Staubli VAL3: AXIS8.pjx

--- AXIS8.pjx ---
Parameters version=s7.2.1 stackSize=5000 millimeterUnit=true
Program file=del.pgx
Program file=find.pgx
Program file=findValue.pgx
Program file=get.pgx
Program file=getSize.pgx
Program file=getType.pgx
Program file=getValue.pgx
Program file=getVelocity.pgx
Program file=loadCycle.pgx
Program file=new.pgx
Program file=onEdit.pgx
Program file=onInsert.pgx
Program file=onProgEnd.pgx
Program file=onRun.pgx
Program file=onStart.pgx
Program file=onStop.pgx
Program file=set.pgx
Program file=setValue.pgx
Program file=setVelocity.pgx
Data file=AXIS8.dtx
Library alias=language path=Disk://kernel/language/language.pjx
Library alias=use path=Disk://kernel/userPage/userPage.pjx

--- AXIS8.dtx ---
num i = 6
public num nSaveaxis = 17746
public num nSaveaxis1 = 55156
public num nVelocity = 8
string l_sItem = "workPos"
public string sItems
public string sSaveaxis = "workPos"
public bool bAxisRun
public aio MbAI_a8Axispose = {link=ModbusSrv-0\Modbus-Word\MbAI_a8Axispose}
public aio MbAI_aCurPosH = {link=ModbusSrv-0\Modbus-Word\MbAI_aCurPosH}
public aio MbAI_aCurPosL = {link=ModbusSrv-0\Modbus-Word\MbAI_aCurPosL}
public aio MbAI_aUnused4 = {link=ModbusSrv-0\Modbus-Word\MbAI_aUnused4}
public aio MbAI_b8MotorErr = {link=ModbusSrv-0\Modbus-Word\MbAI_b8MotorError}
public aio MbAI_b8MotorPow = {link=ModbusSrv-0\Modbus-Word\MbAI_b8MotorPower}
public aio MbAI_bAxis7Reac = {link=ModbusSrv-0\Modbus-Word\MbAI_bAxis7Reached}
public aio MbAI_bAxis8Reac = {link=ModbusSrv-0\Modbus-Word\MbAI_bAxis8Reached}
public aio MbAI_bBackHome = {link=ModbusSrv-0\Modbus-Word\MbAI_bBackHome}
public aio MbAI_bDownLimit = {link=ModbusSrv-0\Modbus-Word\MbAI_bDownLimit}
public aio MbAI_bEndCycl = {link=ModbusSrv-0\Modbus-Word\MbAI_bEndCycl}
public aio MbAI_bHomeDone = {link=ModbusSrv-0\Modbus-Word\MbAI_bHomeDone}
public aio MbAI_bHomeLimit = {link=ModbusSrv-0\Modbus-Word\MbAI_bHomeLimit}
public aio MbAI_bIsHome = {link=ModbusSrv-0\Modbus-Word\MbAI_bIsHome}
public aio MbAI_bMotorErro = {link=ModbusSrv-0\Modbus-Word\MbAI_bMotorError}
public aio MbAI_bMotorPowe = {link=ModbusSrv-0\Modbus-Word\MbAI_bMotorPower}
public aio MbAI_bOutAlarm = {link=ModbusSrv-0\Modbus-Word\MbAI_bOutAlarm}
public aio MbAI_bPowerOn = {link=ModbusSrv-0\Modbus-Word\MbAI_bPowerOn}
public aio MbAI_bStartCycl = {link=ModbusSrv-0\Modbus-Word\MbAI_bStartCycl}
public aio MbAI_bUnused1 = {link=ModbusSrv-0\Modbus-Word\MbAI_bUnused1}
public aio MbAI_bUnused2 = {link=ModbusSrv-0\Modbus-Word\MbAI_bUnused2}
public aio MbAI_bUnused3 = {link=ModbusSrv-0\Modbus-Word\MbAI_bUnused3}
public aio MbAI_bUnused5 = {link=ModbusSrv-0\Modbus-Word\MbAI_bUnused5}
public aio MbAI_bUnused6 = {link=ModbusSrv-0\Modbus-Word\MbAI_bUnused6}
public aio MbAI_bUnused7 = {link=ModbusSrv-0\Modbus-Word\MbAI_bUnused7}
public aio MbAI_bUnused8 = {link=ModbusSrv-0\Modbus-Word\MbAI_bUnused8}
public aio MbAI_bUnused9 = {link=ModbusSrv-0\Modbus-Word\MbAI_bUnused9}
public aio MbAI_bUnused10 = {link=ModbusSrv-0\Modbus-Word\MbAI_bUnused10}
public aio MbAI_bUnused11 = {link=ModbusSrv-0\Modbus-Word\MbAI_bUnused11}
public aio MbAI_bUpLimit = {link=ModbusSrv-0\Modbus-Word\MbAI_bUpLimit}
public aio MbAO_aAxis7Puls = {link=ModbusSrv-0\Modbus-Word\MbAO_aAxis7Pulse}
public aio MbAO_aAxis8Puls = {link=ModbusSrv-0\Modbus-Word\MbAO_aAxis8Pulse}
public aio MbAO_aJogVelo = {link=ModbusSrv-0\Modbus-Word\MbAO_aJogVelo}
public aio MbAO_aJogVelo8 = {link=ModbusSrv-0\Modbus-Word\MbAO_aJogVelo8}
public aio MbAO_aMoveDis = {link=ModbusSrv-0\Modbus-Word\MbAO_aMoveDis}
public aio MbAO_aMoveDis8 = {link=ModbusSrv-0\Modbus-Word\MbAO_aMoveDis8}
public aio MbAO_aMovePosH = {link=ModbusSrv-0\Modbus-Word\MbAO_aMovePosH}
public aio MbAO_aMovePosH8 = {link=ModbusSrv-0\Modbus-Word\MbAO_aMovePosH8}
public aio MbAO_aMovePosL = {link=ModbusSrv-0\Modbus-Word\MbAO_aMovePosL}
public aio MbAO_aMovePosL8 = {link=ModbusSrv-0\Modbus-Word\MbAO_aMovePosL8}
public aio MbAO_aUnused6 = {link=ModbusSrv-0\Modbus-Word\MbAO_aUnused6}
public aio MbAO_aUnused7 = {link=ModbusSrv-0\Modbus-Word\MbAO_aUnused7}
public aio MbAO_aUnused8 = {link=ModbusSrv-0\Modbus-Word\MbAO_aUnused8}
public aio MbAO_aUnused9 = {link=ModbusSrv-0\Modbus-Word\MbAO_aUnused9}
public aio MbAO_aUnused10 = {link=ModbusSrv-0\Modbus-Word\MbAO_aUnused10}
public aio MbAO_aUnused11 = {link=ModbusSrv-0\Modbus-Word\MbAO_aUnused11}
public aio MbAO_aVelocity = {link=ModbusSrv-0\Modbus-Word\MbAO_aVelocity}
public aio MbAO_aVelocity8 = {link=ModbusSrv-0\Modbus-Word\MbAO_aVelocity8}
public aio MbAO_b7Axis = {link=ModbusSrv-0\Modbus-Word\MbAO_b7Axis}
public aio MbAO_b8Axis = {link=ModbusSrv-0\Modbus-Word\MbAO_b8Axis}
public aio MbAO_bAxis7Dire = {link=ModbusSrv-0\Modbus-Word\MbAO_bAxis7Direction}
public aio MbAO_bAxis7Home = {link=ModbusSrv-0\Modbus-Word\MbAO_bAxis7Home}
public aio MbAO_bAxis8Dire = {link=ModbusSrv-0\Modbus-Word\MbAO_bAxis8Direction}
public aio MbAO_bMoveDir = {link=ModbusSrv-0\Modbus-Word\MbAO_bMoveDir}
public aio MbAO_bMoveDirM = {link=ModbusSrv-0\Modbus-Word\MbAO_bMoveDirM}
public aio MbAO_bMovePos8 = {link=ModbusSrv-0\Modbus-Word\MbAO_bMovePos8}
public aio MbAO_bMoveToPos = {link=ModbusSrv-0\Modbus-Word\MbAO_bMoveToPos}
public aio MbAO_bRecordPos = {link=ModbusSrv-0\Modbus-Word\MbAO_bRecordPos}
public aio MbAO_bResetErr = {link=ModbusSrv-0\Modbus-Word\MbAO_bResetErr}
public aio MbAO_bStopMotor = {link=ModbusSrv-0\Modbus-Word\MbAO_bStopMotor}
public aio MbAO_bUnused1 = {link=ModbusSrv-0\Modbus-Word\MbAO_bUnused1}
public aio MbAO_bUnused2 = {link=ModbusSrv-0\Modbus-Word\MbAO_bUnused2}
public aio MbAO_bUnused3 = {link=ModbusSrv-0\Modbus-Word\MbAO_bUnused3}
public aio MbAO_bUnused4 = {link=ModbusSrv-0\Modbus-Word\MbAO_bUnused4}
public aio MbAO_bUnused5 = {link=ModbusSrv-0\Modbus-Word\MbAO_bUnused5}

--- findValue.pgx ---
public program findValue(string& x_sItem[], num& x_nValue[], num& x_nValue1[])
  local num l_nSize
  local string l_sItem
begin
  //
  // find one item in the list
  //
  call getSize(l_nSize)
  for i=0 to l_nSize
    call get(l_sItem,i)
    if l_sItem==x_sItem
      call getValue(x_nValue,i,x_nValue1)
      return
      //go back
    endIf
  endFor
end

--- getType.pgx ---
program getType(string& x_sType[])
  local num l_nPos
  local string l_sPath
begin
  //
  // get the TypePath, show the name
  //
  l_sPath=libPath()
  do
    l_nPos=find(l_sPath,"/")
    if l_nPos==-1
      l_nPos=find(l_sPath,"\")
    endIf
    if l_nPos!=-1
      l_sPath=right(l_sPath,len(l_sPath)-l_nPos-1)
    endIf
  until l_nPos==-1
  x_sType=l_sPath
end

--- loadCycle.pgx ---
public program loadCycle(string& x_sName[], num& x_nResult[])
begin
  //
  // load the select item for the Cycle in advance
  //
end

--- onEdit.pgx ---
public program onEdit(string& x_sItem[])
  local string l_sItem
  local num l_nValue
  local num l_nValue1
begin
  //
  // compose the string
  // call getType(l_sItem)
  // x_sItem=l_sItem+" ???"
  //
  logMsg("OnEdit")
  call findValue(x_sItem,l_nValue,l_nValue1)
  call use:timerDialog("the value is: "+toString("",l_nValue),2)
end

--- onInsert.pgx ---
public program onInsert(string& x_sItem[])
  local string l_sItem
  local string l_sEvent
  local num l_nSize
  local num l_nKey
begin
  //
  // compose the string
  // call getType(l_sItem)
  // x_sItem=l_sItem+" ???"
  //
  // insert all the saveAxis value from the list
  cls()
  call language:message(l_sEvent,65)
  call use:clear(0,13)
  call use:typeCenter(13,l_sEvent,40,true)
  x_sItem=""
  call use:setSizeList(19,0,19,10)
  call use:listcreate("AXIS8")
  l_nSize=size(nSaveaxis)
  for i=0 to l_nSize-1
    l_sEvent=sSaveaxis[i]
    call use:listadd(l_sEvent)
  endFor
  call use:listupdate(0)
  do
    l_nKey=getKey()
    call use:listevent(l_nKey,i,l_sEvent)
    delay(0)
  until l_nKey==255 or l_nKey==270
  if l_nKey==270
    x_sItem="AXIS8>"+l_sEvent
  endIf
  call use:nullKey(l_nKey)
  delay(0)
end

--- onRun.pgx ---
public program onRun(string& x_sItem[])
  local num l_nValue
  local num l_nValue1
  local num l_nVelocity
begin
  //
  // Done, when you execute it
  //
  ////  call findValue(x_sItem,l_nValue)
  ////  aioSet(io:movePulse,l_nValue)
  ////  io:move=true
  ////  delay(0.5)
  ////  io:move=false
  ////  wait(io:atPosition==true or isKeyPressed(255))

  aioSet(MbAO_aMoveDis,0)
  aioSet(MbAO_bMovePos8,0)
  aioSet(MbAO_b8Axis,1)
  bAxisRun=true
//  aioSet(MbAI_bAxis8Reac,0)
  delay(0.5)
  call findValue(x_sItem,l_nValue,l_nValue1)
  call getVelocity(x_sItem,l_nVelocity)
  l_nVelocity=l_nVelocity*1000/60
  aioSet(MbAO_aMovePosL8,l_nValue)
  aioSet(MbAO_aMovePosH8,l_nValue1)
  aioSet(MbAO_aVelocity8,l_nVelocity)
  aioSet(MbAO_bMovePos8,1)
  delay(0.5)
  wait(aioGet(MbAI_bAxis8Reac)==0)
  wait(aioGet(MbAI_bAxis8Reac)==1 or isKeyPressed(255))
  if isKeyPressed(255)
    //if !cycleStatus:bCycle and !cycleStatus:bSimulation
      if aioGet(MbAO_bStopMotor)==1
        aioSet(MbAO_bStopMotor,0)
        delay(0.2)
        aioSet(MbAO_bStopMotor,1)
        delay(0.2)
      else
        aioSet(MbAO_bStopMotor,1)
        delay(0.4)
        aioSet(MbAO_bStopMotor,0)
      endIf
    //endIf
  endIf
  aioSet(MbAO_bMovePos8,0)
  aioSet(MbAO_b8Axis,0)
  // aioSet(io:MbAI_bAxis7Reac,0)
  bAxisRun=false
end

--- onStart.pgx ---
public program onStart(string& x_sItem[])
begin
  //
  // Done on the start of the kernel
  //
end

--- setValue.pgx ---
public program setValue(num x_nValue, num x_nIndex, num x_nValue1)
begin
  // set the value
  // saveAxis[x_nIndex].nValue=x_nValue
  nSaveaxis[x_nIndex]=x_nValue
  nSaveaxis1[x_nIndex]=x_nValue1
end
